PROGRAM MAIN
VAR
	start: BOOL;
	caseswitch: (prepare, starting, selectmovement);
	lool : T_AmsNetID := 'asdasd';
	ProcessXbox: NT_StartProcess;
	idk : UINT; 	
	displayTest : FB_CXSetTextDisplayUSB := (bExecute := TRUE);
END_VAR

//PrepareAxes();
//HbotForwardKinematics();
//nig(CLK := yee);
//gcodeagent(bExecute := TRUE, bNextLine := yee);
//IF PrepareAxes.switchcase = PrepareAxes.movement THEN
//	;
//END_IF

displayTest(
	bExecute:= , 
	sNetID:= , 
	nPort:= 28928, 
	eMode:= eCX2100_WriteLines, 
	sLine1:= '   Welcome to   ', 
	sLine2:= '   ITAP 2023!   ', 
	nCursorPosX:= , 
	nCursorPosY:= , 
	bBusy=> , 
	bError=> , 
	nErrorID=> );

TcXbox();

//GVL.LimitSwitchX := TcXbox.xBoxController.P_Buttons.bA_Button;
//GVL.LimitSwitchY := TcXbox.xBoxController.P_Buttons.bB_Button;

start := tcXbox.xBoxController.P_Buttons.bStart; //addded 20230711 to avoid the need to use HMI to initialise

CASE caseswitch OF
	starting:
		IF start THEN
			caseswitch := Prepare;
		END_IF
		
	Prepare: 
	PrepareAxes();
	IF PrepareAxes.bDone THEN
		caseswitch := selectmovement;
	END_IF
	
	selectmovement:
		MovementTypeSelector();
		GVL.SafetyRun := TRUE;
		
END_CASE

E_Stop();
LimitSwitches();
//C:\Users\weikoons.BECKHOFF\Downloads\HBot_SelfDefinedKinematics\HBot_SelfDefinedKinematics\Hboy\POUs\MovementType_Teach

//ProcessXbox(PATHSTR := 'C:\Users\MaxwellA.BECKHOFF\Documents\TcXaeShell\HBot_SelfDefinedKinematics\HBot_SelfDefinedKinematics\Hboy\POUs\MovementType_Teach\xboxcontrol.exe', 
					//	DIRNAME := 'C:\Users\MaxwellA.BECKHOFF\Documents\TcXaeShell\HBot_SelfDefinedKinematics\HBot_SelfDefinedKinematics\Hboy\POUs\MovementType_Teach\',
						//COMNDLINE := 'GVL.controller 127.0.0.1.1.1',
						//START := TRUE);

END_PROGRAM

(* stored: Version 1.1.0.1, ProductVersion 3.1.4024.12
   POU MAIN: Id {7da8c431-8202-4409-aca8-a2333df93ba0}, SpecialFunc None *)
